ABB RobotStudio station: Lab1.4_20210903-154242.rsstn

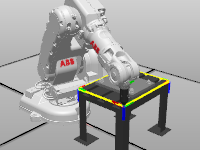
Station Lab1.4 (saved by RobotStudio 21.2.9526.0)
Controller IRB140
  mechanical unit ROB_1: IRB140_6_81_C_03_3, 6 joints, base frame (0, 0, 0) mm
Layout (positions relative to the parent item):
  - IRB140_6_81_C_03_3 [mechanism, from Robots\IRB140_6_81_C_G_03.rslib] at (0, 0, 0) mm; joint values [-0.2552, 0.5481, -0.0658, 0, 1.0885, -0.2552] (rad or m)
  - UISpenholder [mechanism, from RS1\UISpenholder.rslib] at (575, -150, 418) mm, rotated rx -180 ry 0 rz 180 deg
  - table_and_fixture_140 [part, from Training Objects\propeller_table.rslib] at (600, -175, 0) mm, rotated rx 0 ry 0 rz 90 deg
Attachment: UISpenholder is attached to IRB140_6_81_C_03_3 / Link6
Attachment: wobjTable is attached to table_and_fixture_140
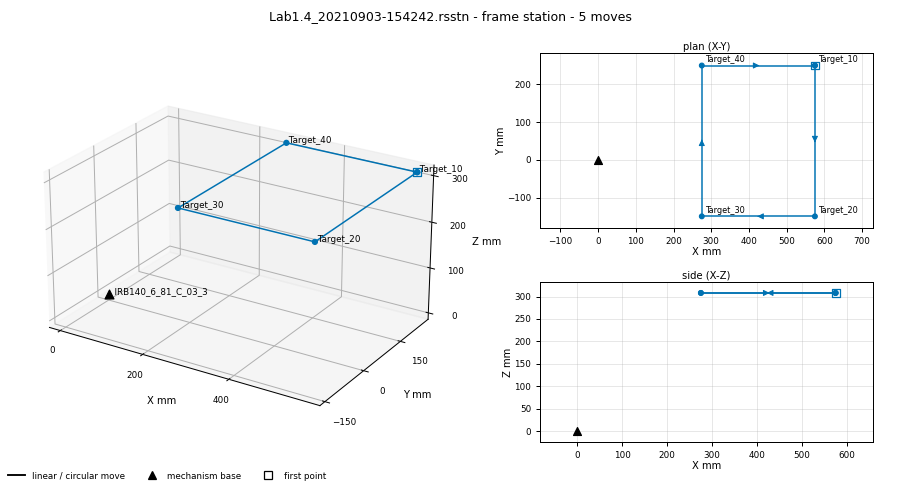
[picture p0: tool path of Lab1.4_20210903-154242.rsstn in frame station, 5 of 5 moves have a stored position in this frame; points joined in program order, loops and branches not executed]
Targets, tools, work objects and paths stored in the station, written as RAPID:
! task T_ROB1
MODULE CalibData
  PERS tooldata UISpenholder:=[TRUE,[[0,0,110],[1,0,0,0]],[1,[0,0,1],[1,0,0,0],0,0,0]];
  TASK PERS wobjdata wobjTable:=[FALSE,TRUE,"",[[425,-575,0],[0.707106781,0,0,0.707106781]],[[425,-150,308],[1,0,0,0]]];
ENDMODULE

! task T_ROB1
MODULE Module1
  CONST robtarget Target_10:=[[400,0,0],[0,0,1,0],[0,0,0,0],[9E+09,9E+09,9E+09,9E+09,9E+09,9E+09]];
  CONST robtarget Target_30:=[[0,300,0],[0,1,0,0],[-1,0,0,0],[9E+09,9E+09,9E+09,9E+09,9E+09,9E+09]];
  CONST robtarget Target_40:=[[400,300,0],[0,-0.707106781,0.707106781,0],[0,0,-2,0],[9E+09,9E+09,9E+09,9E+09,9E+09,9E+09]];
  CONST robtarget Target_20:=[[0,0,0],[0,0.707106781,0.707106781,0],[-1,0,-1,0],[9E+09,9E+09,9E+09,9E+09,9E+09,9E+09]];
  PROC Path_10()
    MoveL Target_10,v1000,z5,UISpenholder\WObj:=wobjTable;
    MoveL Target_20,v1000,z5,UISpenholder\WObj:=wobjTable;
    MoveL Target_30,v1000,z5,UISpenholder\WObj:=wobjTable;
    MoveL Target_40,v1000,z5,UISpenholder\WObj:=wobjTable;
    MoveL Target_10,v1000,z5,UISpenholder\WObj:=wobjTable;
  ENDPROC
ENDMODULE

